{attribute 'enable_dynamic_creation'}	
{attribute 'no_explicit_call' := 'do not call this function block directly'} 
FUNCTION_BLOCK FileTestForEndTask EXTENDS FileContentTask
VAR
	_ClassName : STRING := __POUNAME();

	_TestForEndOfFile : Tc2_System.FB_EOF;
END_VAR

{attribute 'monitoring' := 'call'}
PROPERTY ClassName : STRING
GET
ClassName := _ClassName;
END_GET
END_PROPERTY

METHOD Execute : BOOL
VAR_INPUT
	start : BOOL;
END_VAR
IF start THEN
	Validate();

	_TestForEndOfFile(
		bExecute := FALSE,
		hFile := FilecontentManager.FileHandle,
		sNetId := FilecontentManager.AmsNetId,
		tTimeout := Timeout
	);	
END_IF

_TestForEndOfFile(bExecute := TRUE);

IF _TestForEndOfFile.bError THEN
	//exceptionFactory.ThrowException(__POSITION(), WStringHelper.Concat2("Test for end of file failed", GetErrorMessageByErrorId(_TestForEndOfFile.nErrId)), __POUNAME(), ClassName, CurrentNamespace.Name, __POSITION(), _TestForEndOfFile.nErrId);
ELSIF NOT _TestForEndOfFile.bBusy THEN
	Execute := EXECUTION_STATE.DONE;
END_IF
END_METHOD

PROPERTY IsEndOffile : BOOL
GET
IsEndOffile := _TestForEndOfFile.bEOF;
END_GET
END_PROPERTY

END_FUNCTION_BLOCK

(* stored: Version 1.1.0.1
   POU FileTestForEndTask: Id {fe1ee5b2-a1d2-4d1e-bd5f-c1d42290f541}, SpecialFunc None
   Property ClassName: Id {4f23b7d1-5e36-44ca-8be0-41fdc865291c}
   Get Get: Id {cde6918b-1834-4249-926d-5898a04f481d}
   Method Execute: Id {01a95dd5-7312-4b9e-bd40-af0a6945cbec}
   Property IsEndOffile: Id {de7c80d7-b0ef-48b8-864c-2dfd62ef41ed}
   Get Get: Id {8632d73c-c72d-4377-8610-85866a161051} *)
